SUBAPPLICATION Uebung_003a (* DigitalInput_I1/_I2 auf DigitalOutput_Q1/_I2 *)
  (* Standard: 61499-2; Description: Copyright (c) 2023 Meisterschulen am Ostbahnhof This program and the accompanying materials are made available under the terms of the Eclipse Public License 2.0 which is available at https://www.eclipse.org/legal/epl-2.0/ SPDX-License-Identifier: EPL-2.0 *)
  (* Version 1.0, 2023-10-23, Franz Höpfinger, Meisterschulen am Ostbahnhof *)
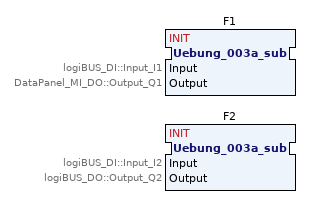
  SUBAPPS
    F1 : Uebung_003a_sub(Input := logiBUS_DI::Input_I1, Output := DataPanel_MI_DO::Output_Q1);
    F2 : Uebung_003a_sub(Input := logiBUS_DI::Input_I2, Output := logiBUS_DO::Output_Q2);
  END_SUBAPPS
END_SUBAPPLICATION
